PROGRAM Pupitre
VAR	
	FB_Fonctions_Pupitre_1:FB_Fonction_Pupitre;
	Cde_en_cours: BOOL;	
END_VAR

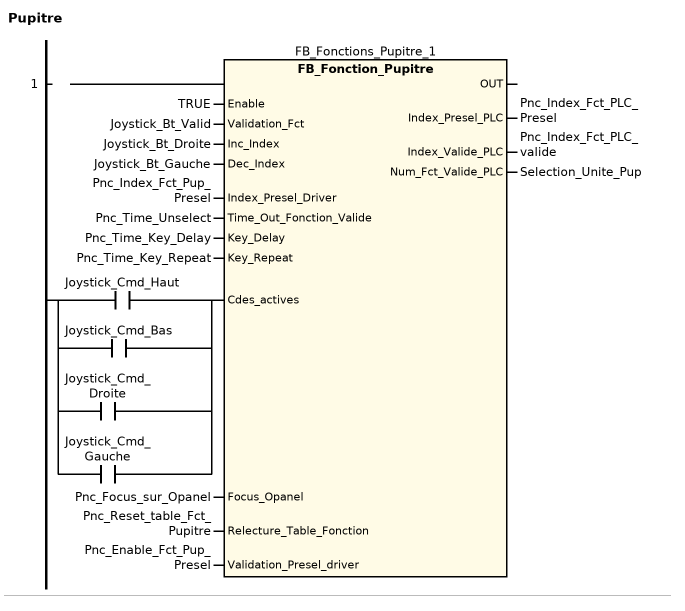
// NETWORK 1
FB_Fonctions_Pupitre_1(
    Enable := TRUE,
    Validation_Fct := Joystick_Bt_Valid,
    Inc_Index := Joystick_Bt_Droite,
    Dec_Index := Joystick_Bt_Gauche,
    Index_Presel_Driver := Pnc_Index_Fct_Pup_Presel,
    Time_Out_Fonction_Valide := Pnc_Time_Unselect,
    Key_Delay := Pnc_Time_Key_Delay,
    Key_Repeat := Pnc_Time_Key_Repeat,
    Cdes_actives := Joystick_Cmd_Haut OR Joystick_Cmd_Bas OR Joystick_Cmd_Droite OR Joystick_Cmd_Gauche,
    Focus_Opanel := Pnc_Focus_sur_Opanel,
    Relecture_Table_Fonction := Pnc_Reset_table_Fct_Pupitre,
    Validation_Presel_driver := Pnc_Enable_Fct_Pup_Presel,
    Index_Presel_PLC => Pnc_Index_Fct_PLC_Presel,
    Index_Valide_PLC => Pnc_Index_Fct_PLC_valide,
    Num_Fct_Valide_PLC => Selection_Unite_Pup); // FB_Fonction_Pupitre

END_PROGRAM

(* stored: Version 1.1.0.1, ProductVersion 3.1.4024.15
   POU Pupitre: Id {f5ad8b2b-411a-4b65-937e-35fde516d2c0}, SpecialFunc None *)
